TYPE (* A Structure with 16 BYTES *)
  (* Version 1.0, 2024-02-21, Franz Höpfinger, HR Agrartechnik GmbH *)
  PACKAGE logiBUS::utils::conversion::types;
  ST32B : STRUCT
    B_00 : BYTE; (* BYTE 00 *)
    B_01 : BYTE; (* BYTE 01 *)
    B_02 : BYTE; (* BYTE 02 *)
    B_03 : BYTE; (* BYTE 03 *)
    B_04 : BYTE; (* BYTE 04 *)
    B_05 : BYTE; (* BYTE 05 *)
    B_06 : BYTE; (* BYTE 06 *)
    B_07 : BYTE; (* BYTE 07 *)
    B_08 : BYTE; (* BYTE 08 *)
    B_09 : BYTE; (* BYTE 09 *)
    B_10 : BYTE; (* BYTE 10 *)
    B_11 : BYTE; (* BYTE 11 *)
    B_12 : BYTE; (* BYTE 12 *)
    B_13 : BYTE; (* BYTE 13 *)
    B_14 : BYTE; (* BYTE 14 *)
    B_15 : BYTE; (* BYTE 15 *)
    B_16 : BYTE; (* BYTE 16 *)
    B_17 : BYTE; (* BYTE 17 *)
    B_18 : BYTE; (* BYTE 18 *)
    B_19 : BYTE; (* BYTE 19 *)
    B_20 : BYTE; (* BYTE 20 *)
    B_21 : BYTE; (* BYTE 21 *)
    B_22 : BYTE; (* BYTE 22 *)
    B_23 : BYTE; (* BYTE 23 *)
    B_24 : BYTE; (* BYTE 24 *)
    B_25 : BYTE; (* BYTE 25 *)
    B_26 : BYTE; (* BYTE 26 *)
    B_27 : BYTE; (* BYTE 27 *)
    B_28 : BYTE; (* BYTE 28 *)
    B_29 : BYTE; (* BYTE 29 *)
    B_30 : BYTE; (* BYTE 30 *)
    B_31 : BYTE; (* BYTE 31 *)
  END_STRUCT;
END_TYPE
